	IF fbWritePar.Error THEN
		nErrorId := UDINT_TO_INT(fbWritePar.ErrorID);
		M_SetError(nErrorId, 'ERROR: Failed to write parameter to Axis');
		// We completed the task (with ERROR) - return TRUE
		nState_PreInit	:= MOTOR_PRE_INIT_STATE_END;
		M_MotorPreInit	:= TRUE;
		RETURN;
	ELSIF fbWritePar.Done THEN
		(* Done! Goto next parameter. *)
		nWriteCounter := nWriteCounter + 1;
		IF nWriteCounter <= 2 THEN
			(* Make the first call with Execute:= FALSE *)
			fbWritePar(	Axis			:= Axis, 
						Execute			:= FALSE, 
						ParameterNumber	:= arrParTableWrite[nWriteCounter].nNumber, 
						Value			:= arrParTableWrite[nWriteCounter].lrValue);
			M_MotorPreInit	:= FALSE;
			RETURN;
		ELSE
			// We completed the task - return TRUE
			nState_PreInit	:= MOTOR_PRE_INIT_STATE_END;
			M_MotorPreInit	:= TRUE;
			RETURN;
		END_IF
	END_IF

	M_MotorPreInit	:= FALSE;
	RETURN;

END_CASE
END_METHOD

(* 
	In this Method we perform all pre-INIT actions like:
	- Disabling axis monitoring limits in order to search for switches without limitations.
	- Reading of Axis parameters, e.g. scale factor.
*) 
METHOD M_MotorReset	: BOOL
VAR_OUTPUT
	nErrorId:	DINT	:= E_MOTOR_ERROR.OK;
END_VAR
VAR_INST
	{attribute 'OPC.UA.DA' := '0'}
	timer_MotorReset:		TON;	(* Timer for measuring duration of events *)
END_VAR
IF nState_Reset = MOTOR_RESET_STATE_END THEN
	M_MotorReset	:= TRUE;
	RETURN;
END_IF

CASE nState_Reset OF
	//////////////////////////
	MOTOR_RESET_STATE_START:
	//////////////////////////
	
// TODO: For now we do SoE Reset every time we INIT an SoE Drive.
// We'll see if we have to do it only if the drive is in error state.
//
//	IF cfg.bSoE_Drive  AND
//		(	((i_nSoE_DriveStatus AND 16#2000) <> 0) OR 
//			((INT_TO_UINT(i_nSoE_PowerStatus) AND 16#0109) <> 16#0009)) THEN

	IF cfg.bSoE_Drive  THEN
		// This is an SoE drive.
		// We have to perform SoE reset that can take up to 10 sec.
		// Goto next state, i.e. SoE Drive Reset 
		nState_Reset	:= MOTOR_RESET_STATE_SoE_RESET;
		M_MotorReset	:= FALSE;
		RETURN;
	ELSE
		// This is an CoE drive.
		// Goto next state, i.e. Reset Axis
		nState_Reset	:= MOTOR_RESET_STATE_RESET_AXIS;
		M_MotorReset	:= FALSE;
		RETURN;
	END_IF
	
	////////////////////////////
	MOTOR_RESET_STATE_SoE_RESET:
	////////////////////////////
	
	// Trigger SoE Drive Reset
	fbSoEReset(Axis := Axis, Execute := FALSE);
	fbSoEReset(Axis := Axis, Execute := TRUE);
	M_SetStatusDescription(E_MOTOR_STATUS.OK, 'Resetting SoE Drive...');
	
	// Restart the 5 sec timer	
	timer_MotorReset(IN:=FALSE);
	timer_MotorReset(IN:=TRUE, PT:=T#10S);
	
	// Goto next state, i.e. Wait for SoE Reset to complete
	nState_Reset	:= MOTOR_RESET_STATE_SoE_WAIT_RESET;
	M_MotorReset	:= FALSE;
	RETURN;

	/////////////////////////////////
	MOTOR_RESET_STATE_SoE_WAIT_RESET:
	/////////////////////////////////
	
	fbSoEReset(Axis := Axis, Execute := TRUE);

	//	If the timeout is detected before RESET is complete, 
	//	then trigger the internal error event. 
	timer_MotorReset();
	IF timer_MotorReset.Q THEN
		timer_MotorReset(IN:=FALSE);	(* Reset the timer *)
		M_SetStatus(E_MOTOR_ERROR.TIMEOUT_RESET);
		nErrorId	:= E_MOTOR_ERROR.TIMEOUT_RESET;
		M_MotorReset:= TRUE;
	END_IF

	(* Check for error or completion *)
	IF fbSoEReset.Error = TRUE THEN
		timer_MotorReset(IN:=FALSE);	(* Reset the timer *)
		IF fbSoEReset.SercosErrId <> 0 THEN
			M_SetError(	E_MOTOR_ERROR.SoE_SERCOS_ERROR, 
						concat('ERROR: SoE Sercos Error #',UINT_TO_STRING(fbSoEReset.SercosErrId)));
			nErrorId	:= UDINT_TO_DINT(fbSoEReset.SercosErrId);
		ELSE
			M_SetError(	E_MOTOR_ERROR.SoE_ADS_ERROR, 
						concat('ERROR: SoE ADS Error #',UINT_TO_STRING(fbSoEReset.AdsErrId)));
			nErrorId	:= UDINT_TO_DINT(fbSoEReset.AdsErrId);
		END_IF
    	fbSoEReset(Axis := Axis, Execute := FALSE);
		nState_Reset	:= MOTOR_RESET_STATE_END;
		M_MotorReset	:= TRUE;
		RETURN; (* goto next cycle *)
	ELSIF NOT fbSoEReset.Busy THEN
		// SoE Reset is complete
    	fbSoEReset(Axis := Axis, Execute := FALSE);
		// Goto next state, i.e. Reset Axis
		nState_Reset	:= MOTOR_RESET_STATE_RESET_AXIS;
		M_MotorReset	:= FALSE;
		RETURN;
 	END_IF

	/////////////////////////////
	MOTOR_RESET_STATE_RESET_AXIS:
	/////////////////////////////
	
	// Reset the motor, i.e. Reset Axis
	fbResetError(Execute:= FALSE, Axis:=Axis);
	fbResetError(Execute:= TRUE,  Axis:=Axis);

	// Restart the 5 sec timer	
	timer_MotorReset(IN:=FALSE);
	timer_MotorReset(IN:=TRUE, PT:=T#5S);
	
	// Goto next state, i.e. Read parameters
	nState_Reset	:= MOTOR_RESET_STATE_WAIT;
	M_MotorReset		:= FALSE;
	RETURN;

	///////////////////////
	MOTOR_RESET_STATE_WAIT:
	///////////////////////
	fbResetError(Execute:= TRUE,  Axis:=Axis);

	//	If the timeout is detected before RESET is complete, 
	//	then trigger the internal error event. 
	timer_MotorReset();
	IF timer_MotorReset.Q THEN
		timer_MotorReset(IN:=FALSE);	(* Reset the timer *)
		M_SetStatus(E_MOTOR_ERROR.TIMEOUT_RESET);
		nErrorId	:= E_MOTOR_ERROR.TIMEOUT_RESET;
		M_MotorReset	:= TRUE;
	END_IF

	(* Check for error or completion *)
	IF fbResetError.Error = TRUE THEN
		timer_MotorReset(IN:=FALSE);	(* Reset the timer *)
		M_SetError(UDINT_TO_INT(fbResetError.ErrorId), M_GetErrorText(UDINT_TO_DINT(fbResetError.ErrorId)));
		nErrorId		:= UDINT_TO_DINT(fbResetError.ErrorId);
		nState_Reset	:= MOTOR_RESET_STATE_END;
		M_MotorReset		:= TRUE;
		RETURN; (* goto next cycle *)
	ELSIF fbResetError.Done = TRUE THEN
		timer_MotorReset(IN:=FALSE);	(* Reset the timer *)
		M_SetStatusDescription(E_MOTOR_STATUS.OK, 'STANDING');
		nState_Reset	:= MOTOR_RESET_STATE_END;
		nErrorId		:= E_MOTOR_ERROR.OK;
		M_MotorReset		:= TRUE;
		RETURN; (* goto next cycle *)
	END_IF

	M_MotorReset	:= FALSE;
	RETURN;

END_CASE
END_METHOD

METHOD M_NormalizePos : LREAL
VAR_INPUT
	lrPos:	LREAL;
END_VAR
M_NormalizePos	:= lrPos;

IF lrPos < 0.0 THEN
	M_NormalizePos	:= lrPos + 360.0;
ELSIF lrPos >= 360.0 THEN
	M_NormalizePos	:= lrPos - 360.0;
END_IF
END_METHOD

METHOD M_NOVRAM_Clear : BOOL
// This method clears SIZEOF(T_MOTOR_CFG) bytes in NOVRAM starting from nNOVRAM_Offset.
// It is needed in cases when the NOVRAM area intended to be used for the motor
// had been previously used for other purpose or it was used with a previous version of T_MOTOR_CFG.
// In these cases the config structure might be corrupt on PLC boot.
// Once the NOVRAM has been cleared, the PLC should be rebooted or "Reset origin" performed.
// M_NOVRAM_Clear() can only be executed in the E_MOTOR_SUBSTATE.NOTOP_NOTREADY state.
VAR_INPUT
	bExecute:	BOOL;
END_VAR
VAR_INST
	{attribute 'OPC.UA.DA' := '0'}
    nMethodState:	INT := 0;	// State Machine current state
	{attribute 'OPC.UA.DA' := '0'}
	nCount:			INT	:= 0;	// Counter for number of cycles to write
END_VAR
// NOVRAM can be cleared only if it is used
IF nNOVRAM_DevId = 0 THEN
	bNOVRAM_Error			:= TRUE;	// Writing to NOVRAM failed
	M_NOVRAM_Clear			:= TRUE;	// Writing to NOVRAM is complete but failed
	M_SetError(E_MOTOR_ERROR.NOVRAM_WRITE, 'Cannot clear NOVRAM. It is not used');
	RETURN;
END_IF

// Check for trigger
IF NOT bExecute THEN
	nMethodState	:= 0;
	nCount			:= 0;
END_IF

// Handle State Machine
CASE nMethodState OF
	0:	// Clear configuration structure
		fbNovReadWrite.bWrite	:= FALSE;	// Go low with Trigger for Write
		fbNovReadWrite.bRead 	:= FALSE;	// bRead will always stay false, i.e. we don't want to read
		bNOVRAM_Error			:= FALSE;	// No error yet
		memset(ADR(stMotorCfg_NOVRAM),0,SIZEOF(stMotorCfg_NOVRAM));	// Clear the CFG structure
		nMethodState 			:= 5;		// Start writing on next call with bExecute=TRUE
		
	5:	// Trigger NOVRAM Write
		fbNovReadWrite.bWrite := TRUE;	// Set Write flag
		nCount	:= nCount + 1;			// Increment counter
		nMethodState := 10;				// Go to next state

	10:	// Check for end of write
		nCount	:= nCount + 1;			// Increment counter
		IF NOT fbNovReadWrite.bBusy THEN
			fbNovReadWrite.bWrite	:= FALSE;	// Stop writing
			nMethodState			:= 0;		// Reset method state
			M_NOVRAM_Clear			:= TRUE;	// Writing NOVRAM is complete
			M_SetStatusDescription(E_MOTOR_STATUS.OK, 'NOVRAM Cleared - Reboot PLC');	// Set status
			RETURN;
		ELSE
			M_SetStatusDescription(E_MOTOR_STATUS.OK, 'Clearing NOVRAM ...');	// Set status
		END_IF
END_CASE


// Perform actual write on every call(while fbNovReadWrite.bWrite = TRUE)
fbNovReadWrite(
	nDevId		:= nNOVRAM_DevId,  
	cbSrcLen	:= SIZEOF(stMotorCfg_NOVRAM), 
	pSrcAddr	:= ADR(stMotorCfg_NOVRAM), 
	nWriteOffs	:= nNOVRAM_Offset, 
	tTimeOut	:= T#5S);

// Check for write errors
IF fbNovReadWrite.bError THEN
	fbNovReadWrite.bWrite	:= FALSE;	// Stop writing
	nMethodState 			:= 0;		// Reset method state
	bNOVRAM_Error			:= TRUE;	// Writing to NOVRAM failed
	M_NOVRAM_Clear			:= TRUE;	// Writing to NOVRAM is complete but failed
	M_SetError(E_MOTOR_ERROR.NOVRAM_WRITE, 'NOVRAM clear failed');
ELSE
	M_NOVRAM_Clear			:= FALSE;	// Writing to NOVRAM has not finished yet
END_IF
END_METHOD

METHOD M_NOVRAM_Load : BOOL
VAR_INPUT
END_VAR
// simple Read / Write to NOVRAM
CASE nNOVRAM_State_R OF
	0:
		fbNovReadWrite.bRead 	:= FALSE;	// Go low with Trigger
		bNOVRAM_Error			:= FALSE;	// Clear error
		nNOVRAM_State_R 		:= 5;		// Goto next state in Reading

	5:
		fbNovReadWrite.bRead	:= TRUE;	// Trigger NOVRAM read 
		nNOVRAM_State_R 		:= 10;

	10:	
		IF NOT fbNovReadWrite.bBusy THEN
			fbNovReadWrite.bRead	:= FALSE;
			nNOVRAM_State_R 		:= 0;
			(* Copy NOVRAM Cfg to motor cfg, after some basic checks. *)
			IF 	stMotorCfg_NOVRAM.lrMaxPosition	>= stMotorCfg_NOVRAM.lrMinPosition THEN
				cfg	:= stMotorCfg_NOVRAM;
			END_IF
			bNOVRAM_Loaded	:= TRUE;	// Loading from NOVRAM is complete
			M_NOVRAM_Load	:= TRUE;	// Return TRUE, i.e. complete
			RETURN;
		END_IF
END_CASE



fbNovReadWrite(
	nDevId		:= nNOVRAM_DevId, 
	cbDestLen	:= SIZEOF(stMotorCfg_NOVRAM), 
	pDestAddr	:= ADR(stMotorCfg_NOVRAM), 
	nReadOffs	:= nNOVRAM_Offset, 
	tTimeOut	:= T#5S, 
	bBusy=> , 
	bError=> , 
	nErrId=> , 
	cbRead=> , 
	cbWrite=> );

IF fbNovReadWrite.bError THEN
	fbNovReadWrite.bRead 	:= FALSE;
	nNOVRAM_State_R 		:= 0;
	bNOVRAM_Error			:= TRUE;	(* Loading from NOVRAM failed *)
	M_NOVRAM_Load			:= TRUE;	(* Loading from NOVRAM is complete but failed *)
ELSE
	M_NOVRAM_Load			:= FALSE;	(* Loading from NOVRAM has not finished yet *)
END_IF
END_METHOD

METHOD M_NOVRAM_Save : BOOL
VAR_INPUT
END_VAR
// Write to NOVRAM
CASE nNOVRAM_State_W OF
	0:
		fbNovReadWrite.bWrite	:= FALSE;	(* Go low with Trigger *)
		bNOVRAM_Error			:= FALSE;
		nNOVRAM_State_W 		:= 5;

	5:
		fbNovReadWrite.bWrite	:= TRUE;	(* Trigger NOVRAM read *)
		nNOVRAM_State_W 		:= 10;

	10:	
		IF NOT fbNovReadWrite.bBusy THEN
			fbNovReadWrite.bWrite	:= FALSE;
			nNOVRAM_State_W			:= 0;
			M_NOVRAM_Save			:= TRUE;	(* Loading from NOVRAM is complete *)
			RETURN;
		END_IF
END_CASE



fbNovReadWrite(
	nDevId		:= nNOVRAM_DevId,
	cbSrcLen	:= SIZEOF(cfg), 
	pSrcAddr	:= ADR(cfg), 
	nWriteOffs	:= nNOVRAM_Offset, 
	tTimeOut	:= T#5S, 
	bBusy=> , 
	bError=> , 
	nErrId=> , 
	cbRead=> , 
	cbWrite=> );

IF fbNovReadWrite.bError THEN
	fbNovReadWrite.bWrite	:= FALSE;
	nNOVRAM_State_W 		:= 0;
	bNOVRAM_Error			:= TRUE;	(* Writing to NOVRAM failed *)
	M_NOVRAM_Save			:= TRUE;	(* Writing to NOVRAM is complete but failed *)
ELSE
	M_NOVRAM_Save			:= FALSE;	(* Writing to NOVRAM has not finished yet *)
END_IF
END_METHOD

METHOD M_SetError
VAR_INPUT
	nErrorCode:	E_MOTOR_ERROR;	// Error number
	sErrorText:	STRING;			// Error text
END_VAR
stat.nStatus		:= E_MOTOR_STATUS.ERROR;
stat.nErrorCode		:= nErrorCode;
stat.sStatus		:= 'ERROR';
stat.sErrorText		:= sErrorText;
END_METHOD

METHOD M_SetRpcStatus : INT
VAR_INPUT
	nErrorCode:	E_MOTOR_RPC_ERROR;
END_VAR
stat.nRpcErrorCode	:= nErrorCode;
stat.sRpcErrorText	:= M_GetRpcErrorText(nErrorCode);

M_SetRpcStatus		:= nErrorCode;
END_METHOD

METHOD M_UpdateSwitches
VAR_INPUT
END_VAR
VAR
	i:			DINT;
	pt:			ARRAY [E_MOTOR_SWITCH_INDEX.LSTOP..E_MOTOR_SWITCH_INDEX.USTOP] OF POINTER TO BOOL;
END_VAR
pt [E_MOTOR_SWITCH_INDEX.LSTOP]	:= ADR(Switches.bLSTOP);
pt [E_MOTOR_SWITCH_INDEX.LHW]		:= ADR(Switches.bLHW);
pt [E_MOTOR_SWITCH_INDEX.REF]		:= ADR(Switches.bREF);
pt [E_MOTOR_SWITCH_INDEX.INDEX]	:= ADR(Switches.bINDEX);
pt [E_MOTOR_SWITCH_INDEX.UHW]		:= ADR(Switches.bUHW);
pt [E_MOTOR_SWITCH_INDEX.USTOP]	:= ADR(Switches.bUSTOP);


FOR i := E_MOTOR_SWITCH_INDEX.LSTOP TO E_MOTOR_SWITCH_INDEX.USTOP DO
	stat.signals[i].bActiveLow	:= cfg.bArrActiveLow[i].bValue;
	stat.signals[i].bActive		:= M_GetLogicalState(pt[i]^, stat.signals[i].bActiveLow);
END_FOR

stat.bStopSwitchNeg	:=	stat.signals[E_MOTOR_SWITCH_INDEX.LSTOP].bActive;
stat.bStopSwitchPos	:=	stat.signals[E_MOTOR_SWITCH_INDEX.USTOP].bActive;
END_METHOD

{attribute 'TcRpcEnable':='1'}
METHOD RPC_Disable : INT
VAR_INPUT
END_VAR
// RPC calls are not allowed in Local mode.
IF stat.bLocal THEN
	RPC_Disable	:= M_SetRpcStatus(E_MOTOR_RPC_ERROR.LOCAL);
	RETURN;
END_IF

// Disable command is accepted only if device is in OP state.
IF stat.nState <> E_MOTOR_STATE.OP THEN
	RPC_Disable	:= M_SetRpcStatus(E_MOTOR_RPC_ERROR.NOT_OP);
	RETURN;
ELSE
	// Set disable command
	ctrl.nCommand := E_MOTOR_COMMAND.DISABLE;
	ctrl.bExecute := TRUE;
	
	// Call was successful
	RPC_Disable	:= M_SetRpcStatus(E_MOTOR_RPC_ERROR.OK);
END_IF
END_METHOD

{attribute 'TcRpcEnable':='1'}
METHOD RPC_Enable : INT
VAR_INPUT
END_VAR
// RPC calls are not allowed in Local mode.
IF stat.bLocal THEN
	RPC_Enable	:= M_SetRpcStatus(E_MOTOR_RPC_ERROR.LOCAL);
	RETURN;
END_IF

// Enable command is accepted only if device is in NOTOP_READY.
IF	stat.nSubstate <> E_MOTOR_SUBSTATE.NOTOP_READY		THEN
	RPC_Enable	:= M_SetRpcStatus(E_MOTOR_RPC_ERROR.NOT_NOTOP_READY);
	RETURN;
ELSE
	// Set enable command
	ctrl.nCommand := E_MOTOR_COMMAND.ENABLE;
	ctrl.bExecute := TRUE;
	
	// Call was successful
	RPC_Enable	:= M_SetRpcStatus(E_MOTOR_RPC_ERROR.OK);
END_IF
END_METHOD

{attribute 'TcRpcEnable':='1'}
METHOD RPC_Init : INT
VAR_INPUT
END_VAR
// If unsafe, INIT is not allowed.
IF NOT in_bSafe THEN
	RPC_Init	:= M_SetRpcStatus(E_MOTOR_RPC_ERROR.UNSAFE);
	RETURN;
END_IF


// RPC calls are not allowed in Local mode.
IF stat.bLocal THEN
	RPC_Init	:= M_SetRpcStatus(E_MOTOR_RPC_ERROR.LOCAL);
	RETURN;
END_IF

// If alredy initialising, then just return OK
IF stat.nSubstate = E_MOTOR_SUBSTATE.NOTOP_INITIALIZING THEN
	RPC_Init	:= M_SetRpcStatus(E_MOTOR_RPC_ERROR.OK);
END_IF

// Init command is accepted only if device is in NOTOP_NOTREADY or ERROR.
IF	stat.nSubstate <> E_MOTOR_SUBSTATE.NOTOP_NOTREADY	AND  
	stat.nSubstate <> E_MOTOR_SUBSTATE.NOTOP_ERROR		THEN
	RPC_Init	:= M_SetRpcStatus(E_MOTOR_RPC_ERROR.NOT_NOTOP_NOTREADY);
	RETURN;
ELSE
	// Set INIT command
	ctrl.nCommand := E_MOTOR_COMMAND.INIT;
	ctrl.bExecute := TRUE;
	
	// Call was successful
	RPC_Init	:= M_SetRpcStatus(E_MOTOR_RPC_ERROR.OK);
END_IF
END_METHOD

{attribute 'TcRpcEnable':='1'}
METHOD RPC_MoveAbs : INT
VAR_INPUT
	in_lrPos:	LREAL;
	in_lrVel:	LREAL;
END_VAR
// If unsafe, move is not allowed.
IF NOT in_bSafe THEN
	RPC_MoveAbs	:= M_SetRpcStatus(E_MOTOR_RPC_ERROR.UNSAFE);
	RETURN;
END_IF

// RPC calls are not allowed in Local mode.
IF stat.bLocal THEN
	RPC_MoveAbs	:= M_SetRpcStatus(E_MOTOR_RPC_ERROR.LOCAL);
	RETURN;
// Move Absolute command is accepted only in OP state.
ELSIF	stat.nState <> E_MOTOR_STATE.OP	THEN
	RPC_MoveAbs	:= M_SetRpcStatus(E_MOTOR_RPC_ERROR.NOT_OP);
	RETURN;
// Set velocity cannot be <=0.0.
ELSIF	in_lrVel <= 0.0	THEN
	RPC_MoveAbs	:= M_SetRpcStatus(E_MOTOR_RPC_ERROR.VEL_NEG);
	RETURN;
// Set velocity cannot be greater than MAX Velocity.
ELSIF	in_lrVel > stat.axis.lrMaxVelocity	THEN
	RPC_MoveAbs	:= M_SetRpcStatus(E_MOTOR_RPC_ERROR.VEL_MAX);
	RETURN;
// If SW limits are active, check the limits
ELSIF cfg.lrMinPosition <> 0.0 OR cfg.lrMaxPosition <> 0.0 THEN
	IF in_lrPos < cfg.lrMinPosition THEN
		RPC_MoveAbs	:= M_SetRpcStatus(E_MOTOR_RPC_ERROR.SW_LIMIT_LOWER);
		RETURN;
	ELSIF in_lrPos > cfg.lrMaxPosition THEN
		RPC_MoveAbs	:= M_SetRpcStatus(E_MOTOR_RPC_ERROR.SW_LIMIT_UPPER);
		RETURN;
	END_IF
END_IF

// Set command
ctrl.nCommand 		:= E_MOTOR_COMMAND.MOTOR_MOVE;
ctrl.nMoveType		:= E_MOTOR_MOVE_TYPE.ABSOLUTE;
ctrl.lrPosition		:= in_lrPos;
ctrl.lrVelocity		:= in_lrVel;
ctrl.bExecute 		:= TRUE;

// Call was successful
RPC_MoveAbs	:= M_SetRpcStatus(E_MOTOR_RPC_ERROR.OK);
END_METHOD

{attribute 'TcRpcEnable':='1'}
METHOD RPC_MoveRel : INT
VAR_INPUT
	in_lrPos:	LREAL;
	in_lrVel:	LREAL;
END_VAR
// If unsafe, move is not allowed.
IF NOT in_bSafe THEN
	RPC_MoveRel	:= M_SetRpcStatus(E_MOTOR_RPC_ERROR.UNSAFE);
	RETURN;
END_IF

// RPC calls are not allowed in Local mode.
IF stat.bLocal THEN
	RPC_MoveRel	:= M_SetRpcStatus(E_MOTOR_RPC_ERROR.LOCAL);
	RETURN;
// Move Relative command is accepted only in OP state.
ELSIF	stat.nState <> E_MOTOR_STATE.OP	THEN
	RPC_MoveRel	:= M_SetRpcStatus(E_MOTOR_RPC_ERROR.NOT_OP);
	RETURN;
// Set velocity cannot be <=0.0.
ELSIF	in_lrVel <= 0.0	THEN
	RPC_MoveRel	:= M_SetRpcStatus(E_MOTOR_RPC_ERROR.VEL_NEG);
	RETURN;
// Set velocity cannot be greater than MAX Velocity.
ELSIF	in_lrVel > stat.axis.lrMaxVelocity	THEN
	RPC_MoveRel	:= M_SetRpcStatus(E_MOTOR_RPC_ERROR.VEL_MAX);
	RETURN;
// If SW limits are active, check the limits
ELSIF cfg.lrMinPosition <> 0.0 OR cfg.lrMaxPosition <> 0.0 THEN
	IF (in_lrPos + stat.lrPosActual) < cfg.lrMinPosition THEN
		RPC_MoveRel	:= M_SetRpcStatus(E_MOTOR_RPC_ERROR.SW_LIMIT_LOWER);
		RETURN;
	ELSIF (in_lrPos + stat.lrPosActual) > cfg.lrMaxPosition THEN
		RPC_MoveRel	:= M_SetRpcStatus(E_MOTOR_RPC_ERROR.SW_LIMIT_UPPER);
		RETURN;
	END_IF
END_IF

// Set command
ctrl.nCommand 		:= E_MOTOR_COMMAND.MOTOR_MOVE;
ctrl.nMoveType		:= E_MOTOR_MOVE_TYPE.RELATIVE;
ctrl.lrOffset		:= in_lrPos;
ctrl.lrVelocity		:= in_lrVel;
ctrl.bExecute 		:= TRUE;

// Call was successful
RPC_MoveRel	:= M_SetRpcStatus(E_MOTOR_RPC_ERROR.OK);
END_METHOD

{attribute 'TcRpcEnable':='1'}
METHOD RPC_MoveVel : INT
VAR_INPUT
	in_lrVel:	LREAL;
END_VAR
// If unsafe, move is not allowed.
IF NOT in_bSafe THEN
	RPC_MoveVel	:= M_SetRpcStatus(E_MOTOR_RPC_ERROR.UNSAFE);
	RETURN;
END_IF

// RPC calls are not allowed in Local mode.
IF stat.bLocal THEN
	RPC_MoveVel	:= M_SetRpcStatus(E_MOTOR_RPC_ERROR.LOCAL);
	RETURN;
END_IF

// Move in Velocity command is accepted only in OP state.
IF	stat.nState <> E_MOTOR_STATE.OP	THEN
	RPC_MoveVel	:= M_SetRpcStatus(E_MOTOR_RPC_ERROR.NOT_OP);
	RETURN;
// Set velocity cannot be 0.0.
ELSIF	in_lrVel = 0.0	THEN
	RPC_MoveVel	:= M_SetRpcStatus(E_MOTOR_RPC_ERROR.VEL_ZERO);
	RETURN;
// Set velocity cannot be greater than MAX Velocity.
// Note that MoveVel() accepts negative velocity. That is
// why we use ABS().
ELSIF	ABS(in_lrVel) > stat.axis.lrMaxVelocity	THEN
	RPC_MoveVel	:= M_SetRpcStatus(E_MOTOR_RPC_ERROR.VEL_MAX);
	RETURN;
ELSE
	// Set command
	ctrl.nCommand 		:= E_MOTOR_COMMAND.MOTOR_MOVE;
	ctrl.nMoveType		:= E_MOTOR_MOVE_TYPE.VELOCITY;
	
	// Set the direction of movement based on the velocity sign.
	// Velocity is always passed as positive.
	IF in_lrVel < 0.0 THEN
		ctrl.lrVelocity		:= -in_lrVel;
		ctrl.nDirection		:= MC_Negative_Direction;
	ELSE
		ctrl.lrVelocity		:= in_lrVel;
		ctrl.nDirection		:= MC_Positive_Direction;
	END_IF

	ctrl.bExecute 		:= TRUE;
	
	// Call was successful
	RPC_MoveVel	:= M_SetRpcStatus(E_MOTOR_RPC_ERROR.OK);
END_IF
END_METHOD

{attribute 'TcRpcEnable':='1'}
METHOD RPC_Reset : INT
VAR_INPUT
END_VAR
// RPC calls are not allowed in Local mode.
IF stat.bLocal THEN
	RPC_Reset	:= M_SetRpcStatus(E_MOTOR_RPC_ERROR.LOCAL);
	RETURN;
END_IF

ctrl.nCommand := E_MOTOR_COMMAND.RESET;
ctrl.bExecute := TRUE;

// Call was successful
RPC_Reset	:= M_SetRpcStatus(E_MOTOR_RPC_ERROR.OK);
END_METHOD

{attribute 'TcRpcEnable':='1'}
METHOD RPC_SetDebug : INT
VAR_INPUT
	in_bDebug:	BOOL 	:= FALSE;		// If TRUE, show event logs of Debug type
END_VAR
// Enable/disable Debugging
cfg.bDebug	:= in_bDebug;

// Call was successful
RPC_SetDebug	:= M_SetRpcStatus(E_MOTOR_RPC_ERROR.OK);
END_METHOD

{attribute 'TcRpcEnable':='1'}
METHOD RPC_SetLog : INT
VAR_INPUT
	in_bLog:	BOOL 	:= FALSE;		// If TRUE, activate event logging
END_VAR
// Enable/disable Logging
cfg.bLog	:= in_bLog;

// Call was successful
RPC_SetLog	:= M_SetRpcStatus(E_MOTOR_RPC_ERROR.OK);
END_METHOD

{attribute 'TcRpcEnable':='1'}
METHOD RPC_Stop : INT
VAR_INPUT
END_VAR
// RPC calls are not allowed in Local mode.
IF stat.bLocal THEN
	RPC_Stop	:= M_SetRpcStatus(E_MOTOR_RPC_ERROR.LOCAL);
	RETURN;
END_IF

ctrl.nCommand := E_MOTOR_COMMAND.STOP;
ctrl.bExecute := TRUE;

// Call was successful
RPC_Stop	:= M_SetRpcStatus(E_MOTOR_RPC_ERROR.OK);
END_METHOD

METHOD UserPostInit : BOOL
VAR_OUTPUT
	nErrorId:	E_MOTOR_ERROR	:= E_MOTOR_ERROR.OK;
END_VAR
VAR
END_VAR
// TODOUSER:
// Dummy implementation.
// Configure cfg.bExecUserPostInit to TRUE.
// Implement PostInit logic.
// If error, set error description in this method using M_SetError(nErrorId, ...) - see below.

stat.sStatus	:= 'User Post-Init Method';

IF Dummy_UserExample() THEN
	UserPostInit	:= TRUE;
	stat.sStatus	:= 'OK';
	RETURN;
END_IF

// Check if the timer has expired. If yes, we have a problem *)
toutCmd();
IF toutCmd.Q = TRUE THEN
	toutCmd(IN := FALSE);
	nErrorId := E_MOTOR_ERROR.TIMEOUT_USER_POSTINIT;
	M_SetError(nErrorId, 'ERROR: Timeout during USER POST INIT');
	UserPostInit	:= TRUE;	// Exit (with error)
	RETURN;
END_IF


(* Check for motion errors *)
IF Axis.Status.Error THEN
	nErrorId	:= UDINT_TO_INT(Axis.Status.ErrorID);
	M_SetError(nErrorId, 'ERROR: Axis error during USER POST INIT');
	UserPostInit	:= TRUE;	// Exit (with error)
	RETURN;
END_IF

// Dummy implementation.
// Dummy error for testing.
//nErrorId := E_MOTOR_ERROR.TIMEOUT;
//M_SetError(nErrorId, 'ERROR: Dummy error during USER POST INIT');
//UserPostInit	:= TRUE;
RETURN;
END_METHOD

METHOD UserPostMove : BOOL
VAR_OUTPUT
	nErrorId:	E_MOTOR_ERROR	:= E_MOTOR_ERROR.OK;
END_VAR
VAR
END_VAR
// TODOUSER:
// Dummy implementation.
// Configure cfg.bExecUserPostMove to TRUE.
// Implement PostMove logic.
// If error, set error description in this method using M_SetError(nErrorId, ...) - see below.

stat.sStatus	:= 'User Post-Move Method';

IF Dummy_UserExample() THEN
	UserPostMove	:= TRUE;
	stat.sStatus	:= 'OK';
	RETURN;
END_IF

// Check if the timer has expired. If yes, we have a problem *)
toutCmd();
IF toutCmd.Q = TRUE THEN
	toutCmd(IN := FALSE);
	nErrorId := E_MOTOR_ERROR.TIMEOUT_USER_POSTMOVE;
	M_SetError(nErrorId, 'ERROR: Timeout during USER POST MOVE');
	UserPostMove	:= TRUE;	// Exit (with error)
	RETURN;
END_IF


(* Check for motion errors *)
IF Axis.Status.Error THEN
	nErrorId	:= UDINT_TO_INT(Axis.Status.ErrorID);
	M_SetError(nErrorId, 'ERROR: Axis error during USER POST MOVE');
	UserPostMove	:= TRUE;	// Exit (with error)
	RETURN;
END_IF

// Dummy implementation.
// Dummy error for testing.
//nErrorId := E_MOTOR_ERROR.TIMEOUT;
//M_SetError(nErrorId, 'ERROR: Dummy error during USER POST MOVE');
//UserPostMove	:= TRUE;
RETURN;
END_METHOD

METHOD UserPreInit : BOOL
VAR_OUTPUT
	nErrorId:	E_MOTOR_ERROR	:= E_MOTOR_ERROR.OK;
END_VAR
VAR
END_VAR
// TODOUSER:
// Dummy implementation.
// Configure cfg.bExecUserPreInit to TRUE.
// Implement PreInit logic.
// If error, set error description in this method using M_SetError(nErrorId, ...) - see below.

stat.sStatus	:= 'User Pre-Init Method';

IF Dummy_UserExample() THEN
	UserPreInit	:= TRUE;
	stat.sStatus	:= 'OK';
	RETURN;
END_IF

// Check if the timer has expired. If yes, we have a problem *)
toutCmd();
IF toutCmd.Q = TRUE THEN
	toutCmd(IN := FALSE);
	nErrorId := E_MOTOR_ERROR.TIMEOUT_USER_PREINIT;
	M_SetError(nErrorId, 'ERROR: Timeout during USER PRE INIT');
	UserPreInit	:= TRUE;	// Exit (with error)
	RETURN;
END_IF


(* Check for motion errors *)
IF Axis.Status.Error THEN
	nErrorId	:= UDINT_TO_INT(Axis.Status.ErrorID);
	M_SetError(nErrorId, 'ERROR: Axis error during USER PRE INIT');
	UserPreInit	:= TRUE;	// Exit (with error)
	RETURN;
END_IF

// Dummy implementation.
// Dummy error for testing.
//nErrorId := E_MOTOR_ERROR.TIMEOUT;
//M_SetError(nErrorId, 'ERROR: Dummy error during USER PRE INIT');
//UserPreInit	:= TRUE;
RETURN;
END_METHOD

METHOD UserPreMove : BOOL
VAR_OUTPUT
	nErrorId:	E_MOTOR_ERROR	:= E_MOTOR_ERROR.OK;
END_VAR
VAR
END_VAR
// TODOUSER:
// Dummy implementation.
// Configure cfg.bExecUserPreMove to TRUE.
// Implement PreMove logic.
// If error, set error description in this method using M_SetError(nErrorId, ...) - see below.

stat.sStatus	:= 'User Pre-Move Method';

IF Dummy_UserExample() THEN
	UserPreMove		:= TRUE;
	stat.sStatus	:= 'OK';
	RETURN;
END_IF

// Check if the timer has expired. If yes, we have a problem *)
toutCmd();
IF toutCmd.Q = TRUE THEN
	toutCmd(IN := FALSE);
	nErrorId := E_MOTOR_ERROR.TIMEOUT_USER_PREMOVE;
	M_SetError(nErrorId, 'ERROR: Timeout during USER PRE MOVE');
	UserPreMove	:= TRUE;	// Exit (with error)
	RETURN;
END_IF


(* Check for motion errors *)
IF Axis.Status.Error THEN
	nErrorId	:= UDINT_TO_INT(Axis.Status.ErrorID);
	M_SetError(nErrorId, 'ERROR: Axis error during USER PRE MOVE');
	UserPreMove	:= TRUE;	// Exit (with error)
	RETURN;
END_IF

// Dummy implementation.
// Dummy error for testing.
//nErrorId := E_MOTOR_ERROR.TIMEOUT;
//M_SetError(nErrorId, 'ERROR: Dummy error during USER PRE MOVE');
//UserPreMove	:= TRUE;
RETURN;
END_METHOD

END_FUNCTION_BLOCK

(* stored: Version 1.1.0.1, ProductVersion 3.1.4024.12
   POU FB_MOTOR: Id {1cb0f4e0-da22-4f09-b830-732d2f4f14b3}, SpecialFunc None
   Method ActionClearNOVRAM: Id {e17cceba-794a-486b-a5fb-702ba675a5f7}
   Method ActionErrExecute: Id {0538174f-0d99-4308-8cd0-823031a574c6}
   Method ActionInitAbort: Id {0676d44b-8c18-48a2-bd40-3a1395654ef7}
   Method ActionInitComplete: Id {07808e00-f135-4349-b4bf-d79495fd33a5}
   Method ActionInitExecute: Id {97b3cbdb-2a31-4af5-89ec-31cfa4270810}
   Method ActionInitReject: Id {f426e1e9-89fa-457d-b49c-9506f6d8243a}
   Method ActionMoveExecute: Id {7440fc23-3594-4859-bb19-bfa09ef5d487}
   Method ActionResetExecute: Id {c1b4383d-ea91-4237-9ab6-5bd638c3c0d1}
   Method ActionSetPosition: Id {9635c4b4-60cf-4dec-8d0a-ac1ca4e6fb2b}
   Method ActionStopExecute: Id {1d1b4441-dc1f-4a25-ae64-afab9af898ea}
   Method ActionUnexpExecute: Id {7fdbcc8b-abb1-4ec9-b1f5-edfef2cce909}
   Method ActivityClearingNOVRAM: Id {14c92b4a-e95a-4615-981a-e8b6e1f06bdf}
   Method ActivityInitAborting: Id {79de9fab-99e6-473d-a7ef-0d52656bc9b3}
   Method ActivityInitializing: Id {8da8ed92-ba64-4e29-a504-03b8696318bd}
   Method ActivityMoving: Id {0aff2a37-5595-4d7e-bb87-d387b85c7afa}
   Method ActivitySettingPosition: Id {b4ec2a0f-c300-4aed-99b2-37ceba3d7026}
   Method ActivityStopping: Id {73143792-fdc5-42e3-922f-9b539cc0c0d7}
   Method CheckForEvents: Id {1bcb3be0-13a0-4554-b509-be6652ab20ef}
   Method Dummy_UserExample: Id {d20f7194-4652-4c55-80c8-c68a3f9ce945}
   Method M_Configure: Id {bd336feb-f03a-429f-92a9-35a747dfe0f6}
   Method M_GetActualPos: Id {08566511-368d-45ab-b69a-734452c5063a}
   Method M_GetOptimisedDistance: Id {758134dc-83ef-4900-b003-f98689075b47}
   Method M_GetOptimisedPosition: Id {5b525718-45b6-4a8f-af78-376d73708e7f}
   Method M_GetRpcErrorText: Id {a6395d91-813f-4cab-a494-3e3d4e48bd2a}
   Method M_HandleEnabled: Id {6ddfffaf-e9d2-4488-9507-44c60001d2ff}
   Method M_MotorBrakeControl: Id {def63cc8-2c88-400d-a379-543e204e8930}
   Method M_MotorInitLock: Id {b6d5b044-a080-4ae1-a4dd-c0f07fcc4062}
   Method M_MotorInitSeq: Id {e4b73036-98b4-40a4-9155-86dc223a113c}
   Method M_MotorPostInit: Id {dbacb6b7-77ef-4d04-bb56-b632330dd2ea}
   Method M_MotorPreInit: Id {30503645-b45e-4cf7-bbf6-7995f6e8e768}
   Method M_MotorReset: Id {ba59baea-f3f0-4813-bfe8-6768cc20f0c4}
   Method M_NormalizePos: Id {6c7349a8-2ea4-4b45-941a-fed8cbce2730}
   Method M_NOVRAM_Clear: Id {affa75df-f26d-48c7-8688-babebcaf23b5}
   Method M_NOVRAM_Load: Id {0e685cc4-2425-4745-aa2a-11da45fc8fa6}
   Method M_NOVRAM_Save: Id {8a81a1d0-fdc1-4739-a174-b649132a747b}
   Method M_SetError: Id {aa3c76d5-5e6f-4703-9b55-28ae4791a991}
   Method M_SetRpcStatus: Id {8fc853df-88b2-40ab-99ba-2b788cf16ba9}
   Method M_UpdateSwitches: Id {1e91313e-c01c-41fb-bbae-73a3c947ff9f}
   Method RPC_Disable: Id {60466611-4f84-4632-bec6-707cbadd749d}
   Method RPC_Enable: Id {4d9488e9-b083-4821-aa71-d9c5fd8da4b8}
   Method RPC_Init: Id {aae974ee-71ef-440d-920b-33456756aa63}
   Method RPC_MoveAbs: Id {aba17171-3ae5-45f9-bc45-4035bb8f1d6b}
   Method RPC_MoveRel: Id {7b854f00-a34d-4806-b1cf-a758f01ba3eb}
   Method RPC_MoveVel: Id {20215d79-9849-4acf-aee6-fa2b1aa10640}
   Method RPC_Reset: Id {009bb7f2-47b9-4dea-b080-934391fea01c}
   Method RPC_SetDebug: Id {6040db75-ab4c-46c7-98e4-7457ef13f944}
   Method RPC_SetLog: Id {43bfa140-8be5-4a9c-bdd7-b6149496dbd5}
   Method RPC_Stop: Id {b2dd7536-18fe-40cb-90c1-82c88b5daf9d}
   Method UserPostInit: Id {c1fca35b-ad64-4254-aaaa-a016bc9a194c}
   Method UserPostMove: Id {7ad8c104-4959-4c28-a7ed-59da6990f786}
   Method UserPreInit: Id {7cdc9816-a2e2-4ed0-b285-2338cb2f22df}
   Method UserPreMove: Id {b6f259c5-41be-47a7-ab14-49f988902160} *)
